INTERFACE I_DriveInverter EXTENDS I_DriveReverse

PROPERTY DeviceData : ST_Inverter
GET
END_GET
END_PROPERTY

PROPERTY InstanceCounter : INT
GET
END_GET
END_PROPERTY

METHOD Reset : BOOL
VAR_INPUT
END_VAR
END_METHOD

METHOD SetSpeed : BOOL
VAR_INPUT
	_speed : REAL;
END_VAR
END_METHOD

END_INTERFACE

(* stored: Version 1.1.0.1, ProductVersion 3.1.4024.12
   Itf I_DriveInverter: Id {9a5e992e-1284-4147-ba3f-8a6070e5989f}
   Property DeviceData: Id {1eaa2b74-a49a-4ae6-8a07-2d855495bacf}
   Get Get: Id {c3d1219e-a4f9-425f-94f8-da59e4e8a604}
   Property InstanceCounter: Id {ad8649c7-fdbd-40d3-b7cc-aa849d0ab7e0}
   Get Get: Id {0e93bed3-4072-4dd2-870f-572b7e9fe37d}
   Method Reset: Id {858c975f-f164-483b-b967-bc1f72971972}
   Method SetSpeed: Id {f2796ee0-7648-4000-afac-c6ef6a0549fc} *)
